{attribute 'qualified_only'}
{attribute 'strict'}
TYPE ST_SysPar :
STRUCT
	sRemoteHost			: T_IPv4Addr ;
	nRemotePort			: UINT := 0;    
	bySlaveID 			: BYTE;	
END_STRUCT
END_TYPE

(* stored: Version 1.1.0.1, ProductVersion 3.1.4024.9
   DUT ST_SysPar: Id {45ffb368-a3c9-4b37-a507-3ff1a3b3674a} *)
